Staubli VAL3: ThrottleLogMsg.pjx

--- ThrottleLogMsg.pjx ---
Parameters version=s7.7.2 stackSize=5000 millimeterUnit=true
Program file=start.pgx
Program file=stop.pgx
Data file=ThrottleLogMsg.dtx

--- ThrottleLogMsg.dtx ---
public string sMsg
public num nSeverity
public num nLastLogTime
public num nThrottleInterval
public num nMsgCountSinceLastLog
